PROGRAM onOffLed
VAR
    inputSwitch : BOOL;
    outputLED : BOOL;
    rTrig : R_TRIG;
END_VAR

rTrig(CLK:= inputSwitch);

IF rTrig.Q THEN
    outputLED:= NOT outputLED;
END_IF
inputSwitch:= FALSE;

END_PROGRAM

(* stored: Version 1.1.0.1, ProductVersion 3.1.4024.5
   POU onOffLed: Id {b6065991-9aa8-49bd-9736-ef4d1d8a8a69}, SpecialFunc None *)
